Fanuc KAREL source: IO0085.KL

-- PROVISIONAL review KL for V1013-1; original PC SHA256 71f2e2b784c84cf85c3e6d5836aadac1acec03f0552de6d731562cf64da5d582
-- Incomplete behavior may be omitted. Consult companion uncertainty JSON. Do not deploy.
PROGRAM IO0085
%NOLOCKGROUP
-- UNRESOLVED_LOCAL_POOL 5 cells at code offset 13; source declarations unknown
-- DIRECT_LOCAL_WORD_ACCESS alone does not prove INTEGER, REAL, or BOOLEAN
BEGIN
  -- UNRESOLVED_PC offsets 0-18; opcodes 2B,2C,7B
  -- UNRESOLVED_PC offsets 23-30; opcodes 9D,23
  -- UNRESOLVED_PC offsets 35-49; opcodes 2E,22,9D,33,35
  -- UNRESOLVED_PC offsets 54-61; opcodes 9D,23
  -- UNRESOLVED_PC offsets 66-77; opcodes 2E,23
  -- UNRESOLVED_PC offsets 82-97; opcodes 21,19,9C,5B,79
  -- UNRESOLVED_PC offsets 102-116; opcodes 21,9D,52,23
  -- UNRESOLVED_PC offsets 126-130; opcodes 7F
  -- UNRESOLVED_PC offsets 135-139; opcodes 27,AA
  -- UNRESOLVED_PC offsets 144-148; opcodes 7F
END IO0085
